// TIA Portal V15.1 export
// export: Created 2024-06-21T08:40:59.9132549Z, ExportSetting WithDefaults, DisplayName Totally Integrated Automation Portal, DisplayVersion V15.1 Update 5, DisplayName TIA Portal Openness, DisplayVersion V15.1 Update 5, DisplayName SINAMICS Startdrive Advanced, DisplayVersion V15.1, DisplayName G130, G150, S120, S150, SINAMICS MV, S210, DisplayVersion V15.1, DisplayName G110M, G120, G120C, G120D, G120P, DisplayVersion V15.1, DisplayName STEP 7 Professional, DisplayVersion V15.1 Update 5, DisplayName STEP 7 Safety, DisplayVersion V15.1, DisplayName WinCC Professional, DisplayVersion V15.1 Update 5, DisplayName SIMATIC Visualization Architect, DisplayVersion V15.1
FUNCTION_BLOCK "LPNIODiagHMIS7-1500"   // FB2214, FBD
TITLE = LPNIODiagHMIS7-1500
{ S7_Optimized_Access := 'FALSE' }
VERSION : 0.1
// stored: AutoNumber false, IsIECCheckEnabled false, SetENOAutomatically False, UDAEnableTagReadback false
   VAR_INPUT
      I_DeviceNumber { ExternalAccessible := 'False'; ExternalVisible := 'False'; ExternalWritable := 'False'} : Int;   // Device number in the hardware config
      I_Name { ExternalAccessible := 'False'; ExternalVisible := 'False'; ExternalWritable := 'False'} : String[25];   // Name device from list
      I_IPAddress { ExternalAccessible := 'False'; ExternalVisible := 'False'; ExternalWritable := 'False'} : String[15];   // IP address device from list
      I_MACAddress { ExternalAccessible := 'False'; ExternalVisible := 'False'; ExternalWritable := 'False'} : String[18];   // MAC address device from list
      I_AlarmClass { ExternalAccessible := 'False'; ExternalVisible := 'False'; ExternalWritable := 'False'} : Char;   // Alarm class -> A - B - C - D or E
      I_EnableAlarm { ExternalAccessible := 'False'; ExternalVisible := 'False'; ExternalWritable := 'False'} : Bool := TRUE;   // Enable alarm from upper level
      I_EnableButtons { ExternalAccessible := 'False'; ExternalVisible := 'False'; ExternalWritable := 'False'} : Bool;   // Enable to use the buttons in the pop-up -> "Activate" and "Deactivate"
   END_VAR
   VAR_OUTPUT
      O_Alarm { ExternalAccessible := 'False'; ExternalVisible := 'False'; ExternalWritable := 'False'} : Bool;   // Alarm A
      O_AC_Faulty { ExternalAccessible := 'False'; ExternalVisible := 'False'; ExternalWritable := 'False'} : Bool;   // Device is in faulty
      O_AD_Disabled { ExternalAccessible := 'False'; ExternalVisible := 'False'; ExternalWritable := 'False'} : Bool;   // Device is disabled
      O_AlarmABcondition { ExternalAccessible := 'False'; ExternalVisible := 'False'; ExternalWritable := 'False'} : Bool;   // Alarm AB condition
      H_IAnim { ExternalAccessible := 'False'; ExternalVisible := 'False'; ExternalWritable := 'False'} : Word;   // HMI Animation color of the icon
      H_IAnim2 { ExternalAccessible := 'False'; ExternalVisible := 'False'; ExternalWritable := 'False'} : Int;   // HMI Animation
   END_VAR
   VAR_IN_OUT
      IO_PNIODIAG_Global : "H_PNIODiagS7-1500";
   END_VAR
   VAR DB_SPECIFIC
      H_In : Struct   // HMI
         HMICmd : Word;   // Commands from HMI
         Mode : Int;   // Mode
      END_STRUCT;
      H_Out : Struct   // HMI
         Anim : Word;   // HMI Animation Word
         DeviceNumber : Int;   // HMI Device number (node)
         "Name" : String[25];   // HMI Profinet name
         IPAddress : String[15];   // HMI IP Address
         MACAddress : String[18];   // HMI MAC Address
         DBnr : Int;   // HMI Animation DB number
      END_STRUCT;
      HMICmdActivated { ExternalAccessible := 'False'; ExternalVisible := 'False'; ExternalWritable := 'False'} : Bool;   // HMI Cmd
      HMICmdDeactivated { ExternalAccessible := 'False'; ExternalVisible := 'False'; ExternalWritable := 'False'} : Bool;   // HMI Cmd
      Alarm { ExternalAccessible := 'False'; ExternalVisible := 'False'; ExternalWritable := 'False'} : Bool;   // Alarm
      AlarmClass_A { ExternalAccessible := 'False'; ExternalVisible := 'False'; ExternalWritable := 'False'} : Bool;   // The alarm is from alarm class A
      AlarmClass_B { ExternalAccessible := 'False'; ExternalVisible := 'False'; ExternalWritable := 'False'} : Bool;   // The alarm is from alarm class B
      AlarmClass_C { ExternalAccessible := 'False'; ExternalVisible := 'False'; ExternalWritable := 'False'} : Bool;   // The alarm is from alarm class C
      AlarmClass_D { ExternalAccessible := 'False'; ExternalVisible := 'False'; ExternalWritable := 'False'} : Bool;   // The alarm is from alarm class D
      AlarmClass_E { ExternalAccessible := 'False'; ExternalVisible := 'False'; ExternalWritable := 'False'} : Bool;   // The alarm is from alarm class E
      AlarmCond { ExternalAccessible := 'False'; ExternalVisible := 'False'; ExternalWritable := 'False'} : Bool;   // Alarm condition
      DBnr { ExternalAccessible := 'False'; ExternalVisible := 'False'; ExternalWritable := 'False'} : Int;   // HMI DB number
      DeviceExist { ExternalAccessible := 'False'; ExternalVisible := 'False'; ExternalWritable := 'False'} : Bool;   // Device exist
      DeviceDisabled { ExternalAccessible := 'False'; ExternalVisible := 'False'; ExternalWritable := 'False'} : Bool;   // Device is disabled
      DeviceFaulty { ExternalAccessible := 'False'; ExternalVisible := 'False'; ExternalWritable := 'False'} : Bool;   // Device is in faulty
      DeviceServiceReq { ExternalAccessible := 'False'; ExternalVisible := 'False'; ExternalWritable := 'False'} : Bool;   // Device has a service request
      EnableBtnActivate { ExternalAccessible := 'False'; ExternalVisible := 'False'; ExternalWritable := 'False'} : Bool;   // Enable button in pop-up
      EnableBtnDeactivate { ExternalAccessible := 'False'; ExternalVisible := 'False'; ExternalWritable := 'False'} : Bool;   // Enable button in pop-up
      TimerDeviceDisabled { ExternalAccessible := 'False'; ExternalVisible := 'False'; ExternalWritable := 'False'; S7_SetPoint := 'True'} : TOF_TIME;   // Timer
      TimerActivateDeactivateBusy { ExternalAccessible := 'False'; ExternalVisible := 'False'; ExternalWritable := 'False'; S7_SetPoint := 'True'} : TOF_TIME;   // Timer
      TimerHMICmdActivated { ExternalAccessible := 'False'; ExternalVisible := 'False'; ExternalWritable := 'False'; S7_SetPoint := 'True'} : TON_TIME;   // Timer
      TimerHMICmdDeactivated { ExternalAccessible := 'False'; ExternalVisible := 'False'; ExternalWritable := 'False'; S7_SetPoint := 'True'} : TON_TIME;   // Timer
   END_VAR
BEGIN

NETWORK
TITLE = **** 1 - Inputs **** DB number
// DB number
      L     DINO;
      T     #DBnr;

NETWORK
TITLE = **** 1 - Inputs **** Alarm class
// Alarm class
// Alarm class = E
      L     #I_AlarmClass;
      L     'E';
      ==I;
      =     #AlarmClass_E;

// Alarm class = D
      L     #I_AlarmClass;
      L     'D';
      ==I;
      =     #AlarmClass_D;

// Alarm class = C
      L     #I_AlarmClass;
      L     'C';
      ==I;
      =     #AlarmClass_C;

// Alarm class = B
      L     #I_AlarmClass;
      L     'B';
      ==I;
      =     #AlarmClass_B;

// Alarm class = A
      AN    #AlarmClass_B;
      AN    #AlarmClass_C;
      AN    #AlarmClass_D;
      AN    #AlarmClass_E;
      =     #AlarmClass_A;


REGION Network 3: **** 1 - Inputs **** HMI Cmd
   // Extract HMI Cmd
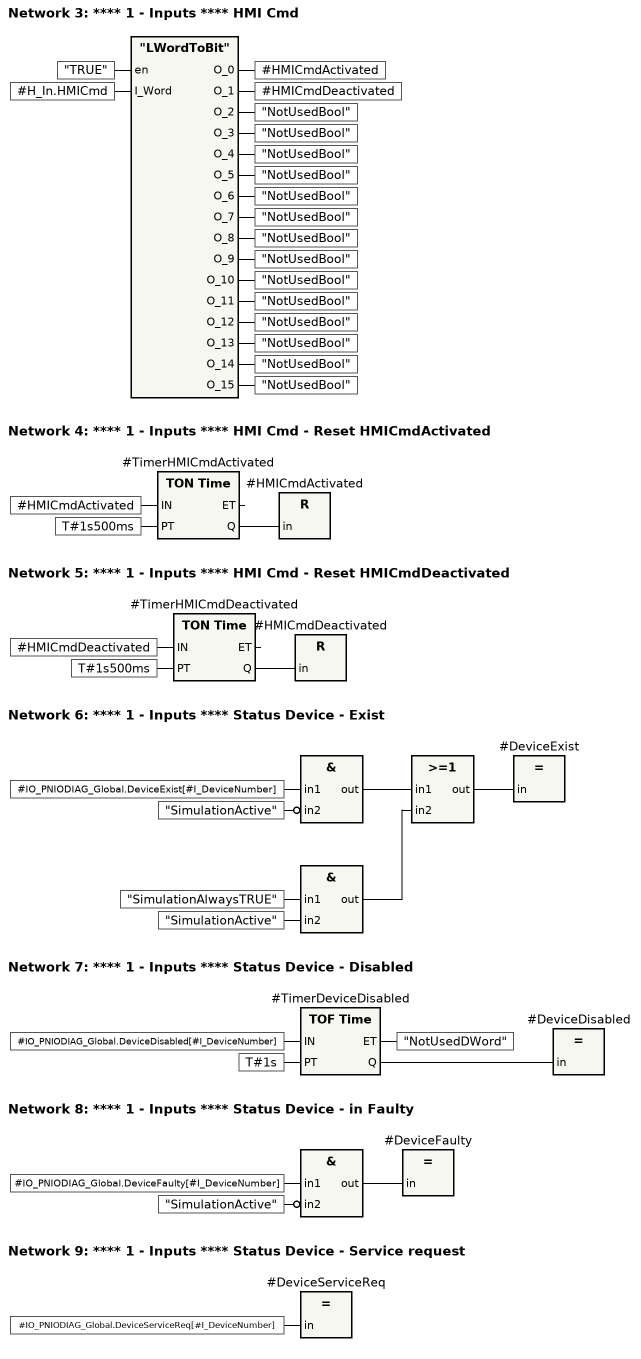
   IF "TRUE" THEN
       "LWordToBit"(I_Word := #H_In.HMICmd,
                    O_0 => #HMICmdActivated,
                    O_1 => #HMICmdDeactivated,
                    O_2 => "NotUsedBool",
                    O_3 => "NotUsedBool",
                    O_4 => "NotUsedBool",
                    O_5 => "NotUsedBool",
                    O_6 => "NotUsedBool",
                    O_7 => "NotUsedBool",
                    O_8 => "NotUsedBool",
                    O_9 => "NotUsedBool",
                    O_10 => "NotUsedBool",
                    O_11 => "NotUsedBool",
                    O_12 => "NotUsedBool",
                    O_13 => "NotUsedBool",
                    O_14 => "NotUsedBool",
                    O_15 => "NotUsedBool");
   END_IF;
END_REGION

REGION Network 4: **** 1 - Inputs **** HMI Cmd - Reset HMICmdActivated
   // HMI Cmd - Reset HMICmdActivated
   #TimerHMICmdActivated(IN := #HMICmdActivated, PT := T#1s500ms);   // TON
   IF #TimerHMICmdActivated.Q THEN #HMICmdActivated := FALSE; END_IF;
END_REGION

REGION Network 5: **** 1 - Inputs **** HMI Cmd - Reset HMICmdDeactivated
   // HMI Cmd - Reset HMICmdDeactivated
   #TimerHMICmdDeactivated(IN := #HMICmdDeactivated, PT := T#1s500ms);   // TON
   IF #TimerHMICmdDeactivated.Q THEN #HMICmdDeactivated := FALSE; END_IF;
END_REGION

REGION Network 6: **** 1 - Inputs **** Status Device - Exist
   // Status Device - Exist
   #DeviceExist := (#IO_PNIODIAG_Global.DeviceExist[#I_DeviceNumber] AND NOT "SimulationActive") OR ("SimulationAlwaysTRUE" AND "SimulationActive");
END_REGION

REGION Network 7: **** 1 - Inputs **** Status Device - Disabled
   // Status Device - Disabled
   #TimerDeviceDisabled(IN := #IO_PNIODIAG_Global.DeviceDisabled[#I_DeviceNumber],   // TOF
                        PT := T#1s,
                        ET => "NotUsedDWord");
   #DeviceDisabled := #TimerDeviceDisabled.Q;
END_REGION

REGION Network 8: **** 1 - Inputs **** Status Device - in Faulty
   // Status Device - in Faulty
   #DeviceFaulty := #IO_PNIODIAG_Global.DeviceFaulty[#I_DeviceNumber] AND NOT "SimulationActive";
END_REGION

REGION Network 9: **** 1 - Inputs **** Status Device - Service request
   // Status Device - Service request
   #DeviceServiceReq := #IO_PNIODIAG_Global.DeviceServiceReq[#I_DeviceNumber];
END_REGION

REGION Network 10: **** 1 - Inputs **** Timer Signal ActivateDeactivateBusy
   // Timer Signal ActivateDeactivateBusy
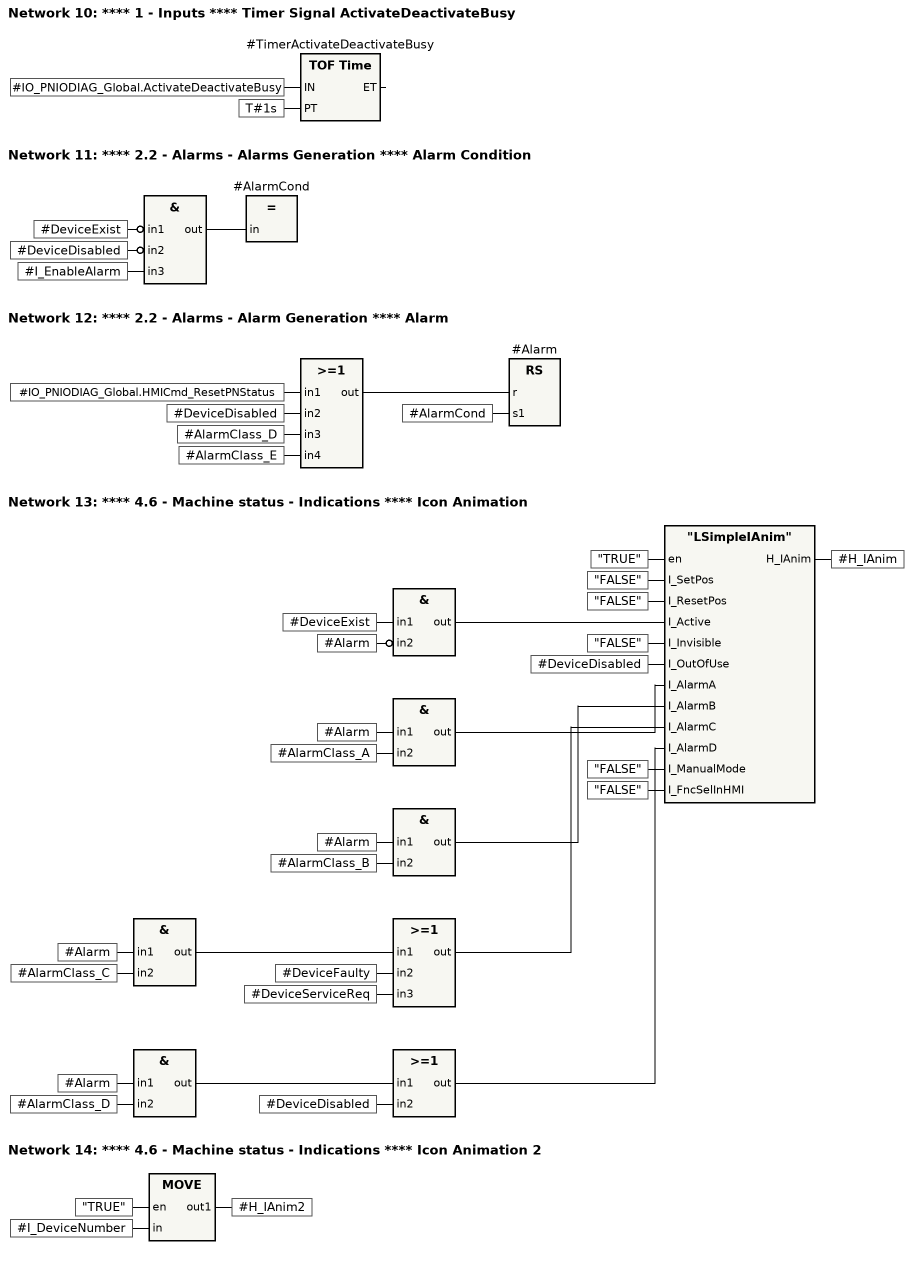
   #TimerActivateDeactivateBusy(IN := #IO_PNIODIAG_Global.ActivateDeactivateBusy, PT := T#1s);   // TOF
END_REGION

REGION Network 11: **** 2.2 - Alarms - Alarms Generation **** Alarm Condition
   // Condition for the Alarm
   #AlarmCond := NOT #DeviceExist AND NOT #DeviceDisabled AND #I_EnableAlarm;
END_REGION

REGION Network 12: **** 2.2 - Alarms - Alarm Generation **** Alarm
   // Alarm
   IF #IO_PNIODIAG_Global.HMICmd_ResetPNStatus OR #DeviceDisabled OR #AlarmClass_D OR #AlarmClass_E THEN
       #Alarm := FALSE;   // RS flip-flop
   END_IF;
   IF #AlarmCond THEN #Alarm := TRUE; END_IF;
END_REGION

REGION Network 13: **** 4.6 - Machine status - Indications **** Icon Animation
   // Icon Animation
   IF "TRUE" THEN
       "LSimpleIAnim"(I_SetPos := "FALSE",
                      I_ResetPos := "FALSE",
                      I_Active := #DeviceExist AND NOT #Alarm,
                      I_Invisible := "FALSE",
                      I_OutOfUse := #DeviceDisabled,
                      I_AlarmA := #Alarm AND #AlarmClass_A,
                      I_AlarmB := #Alarm AND #AlarmClass_B,
                      I_AlarmC := (#Alarm AND #AlarmClass_C) OR #DeviceFaulty OR #DeviceServiceReq,
                      I_AlarmD := (#Alarm AND #AlarmClass_D) OR #DeviceDisabled,
                      I_ManualMode := "FALSE",
                      I_FncSelInHMI := "FALSE",
                      H_IAnim => #H_IAnim);
   END_IF;
END_REGION

REGION Network 14: **** 4.6 - Machine status - Indications **** Icon Animation 2
   // Icon Animation Device number
   IF "TRUE" THEN #H_IAnim2 := #I_DeviceNumber; END_IF;
END_REGION

REGION Network 15: **** 4.6 - Machine status - Indications **** Animation
   // Animation for HMI
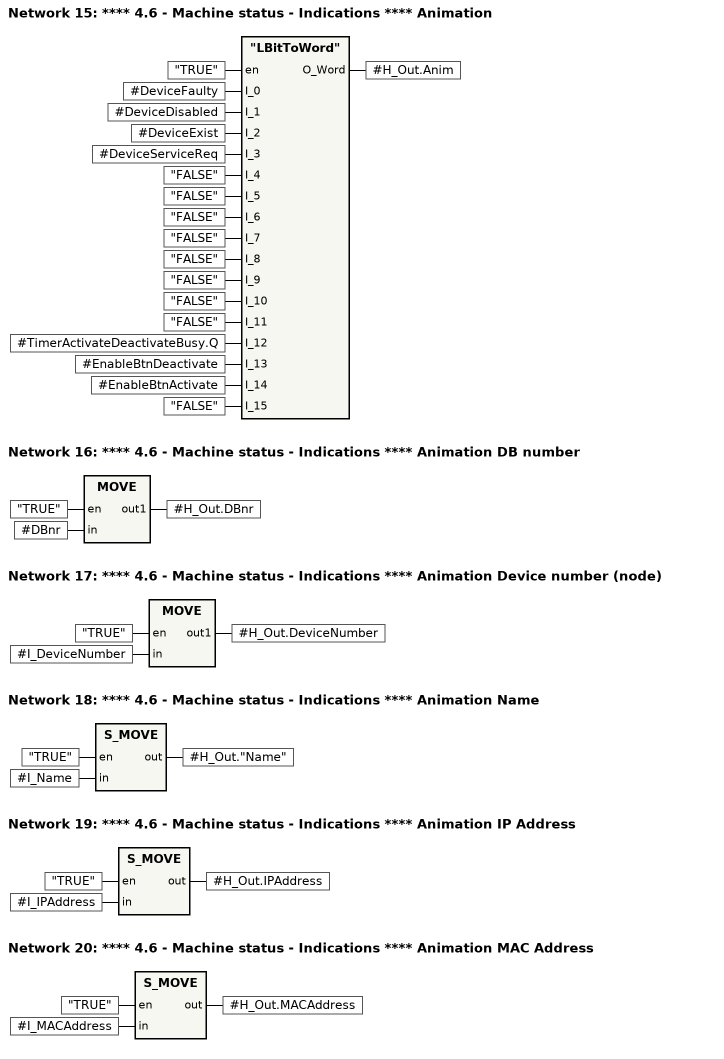
   IF "TRUE" THEN
       "LBitToWord"(I_0 := #DeviceFaulty,
                    I_1 := #DeviceDisabled,
                    I_2 := #DeviceExist,
                    I_3 := #DeviceServiceReq,
                    I_4 := "FALSE",
                    I_5 := "FALSE",
                    I_6 := "FALSE",
                    I_7 := "FALSE",
                    I_8 := "FALSE",
                    I_9 := "FALSE",
                    I_10 := "FALSE",
                    I_11 := "FALSE",
                    I_12 := #TimerActivateDeactivateBusy.Q,
                    I_13 := #EnableBtnDeactivate,
                    I_14 := #EnableBtnActivate,
                    I_15 := "FALSE",
                    O_Word => #H_Out.Anim);
   END_IF;
END_REGION

REGION Network 16: **** 4.6 - Machine status - Indications **** Animation DB number
   // DB number
   IF "TRUE" THEN #H_Out.DBnr := #DBnr; END_IF;
END_REGION

REGION Network 17: **** 4.6 - Machine status - Indications **** Animation Device number (node)
   // Device number (node)
   IF "TRUE" THEN #H_Out.DeviceNumber := #I_DeviceNumber; END_IF;
END_REGION

REGION Network 18: **** 4.6 - Machine status - Indications **** Animation Name
   // Name
   IF "TRUE" THEN #H_Out."Name" := #I_Name; END_IF;
END_REGION

REGION Network 19: **** 4.6 - Machine status - Indications **** Animation IP Address
   // IP Address
   IF "TRUE" THEN #H_Out.IPAddress := #I_IPAddress; END_IF;
END_REGION

REGION Network 20: **** 4.6 - Machine status - Indications **** Animation MAC Address
   // MAC Address
   IF "TRUE" THEN #H_Out.MACAddress := #I_MACAddress; END_IF;
END_REGION

REGION Network 21: **** 5.2 - Equations - Flow **** Activated or Deactived a device to the global FB
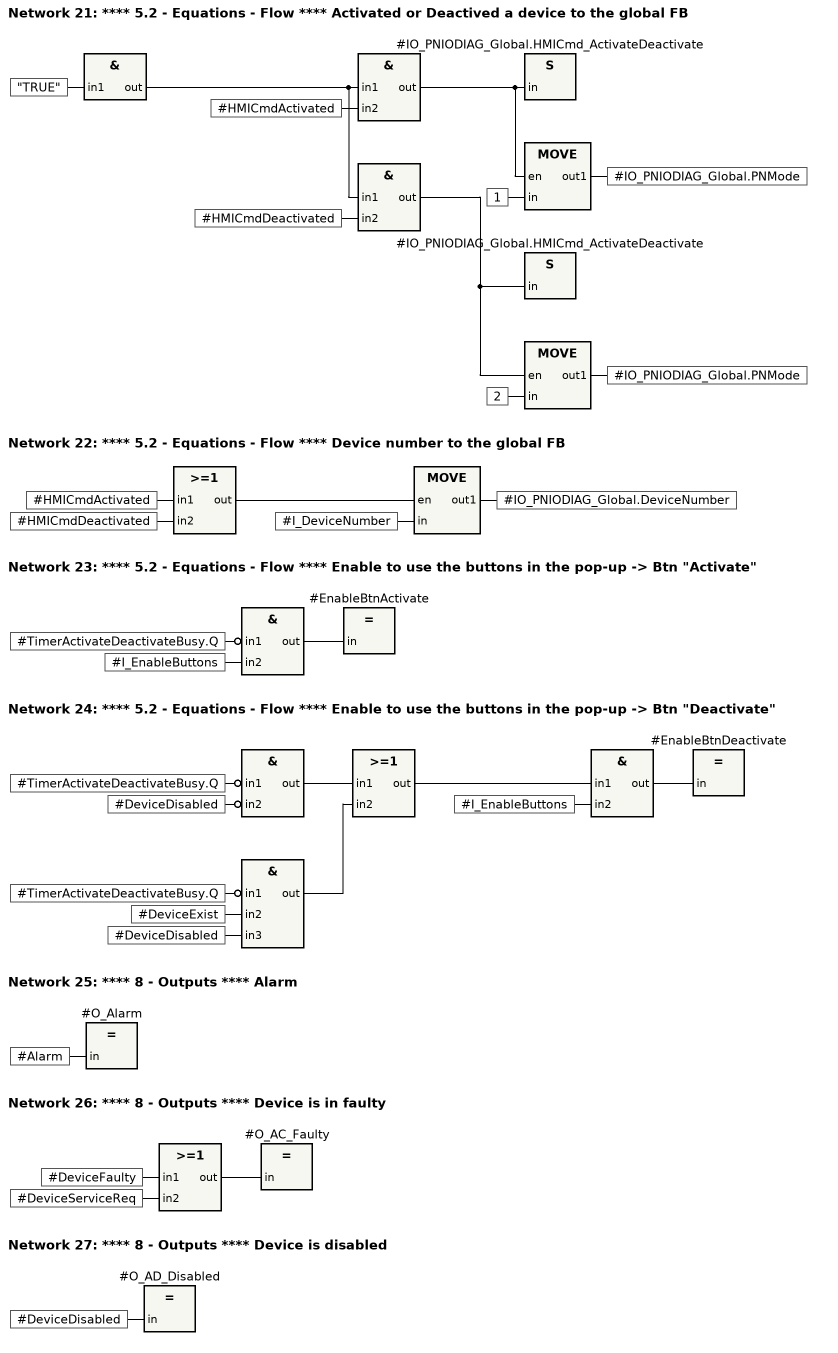
   IF "TRUE" AND #HMICmdActivated THEN
       #IO_PNIODIAG_Global.HMICmd_ActivateDeactivate := TRUE;
       #IO_PNIODIAG_Global.PNMode := 1;
   END_IF;
   IF "TRUE" AND #HMICmdDeactivated THEN
       #IO_PNIODIAG_Global.HMICmd_ActivateDeactivate := TRUE;
       #IO_PNIODIAG_Global.PNMode := 2;
   END_IF;
END_REGION

REGION Network 22: **** 5.2 - Equations - Flow **** Device number to the global FB
   IF #HMICmdActivated OR #HMICmdDeactivated THEN
       #IO_PNIODIAG_Global.DeviceNumber := #I_DeviceNumber;
   END_IF;
END_REGION

REGION Network 23: **** 5.2 - Equations - Flow **** Enable to use the buttons in the pop-up -> Btn "Activate"
   // Enable to use the buttons in the pop-up -> Btn "Activate"
   #EnableBtnActivate := NOT #TimerActivateDeactivateBusy.Q AND #I_EnableButtons;
END_REGION

REGION Network 24: **** 5.2 - Equations - Flow **** Enable to use the buttons in the pop-up -> Btn "Deactivate"
   // Enable to use the buttons in the pop-up -> Btn "Deactivate"
   #EnableBtnDeactivate := ((NOT #TimerActivateDeactivateBusy.Q AND NOT #DeviceDisabled) OR (NOT #TimerActivateDeactivateBusy.Q AND #DeviceExist AND #DeviceDisabled)) AND #I_EnableButtons;
END_REGION

REGION Network 25: **** 8 - Outputs **** Alarm
   // Alarm
   #O_Alarm := #Alarm;
END_REGION

REGION Network 26: **** 8 - Outputs **** Device is in faulty
   #O_AC_Faulty := #DeviceFaulty OR #DeviceServiceReq;
END_REGION

REGION Network 27: **** 8 - Outputs **** Device is disabled
   #O_AD_Disabled := #DeviceDisabled;
END_REGION

REGION Network 28: **** 8 - Outputs **** Alarm AB Condition
   // Alarm AB condition
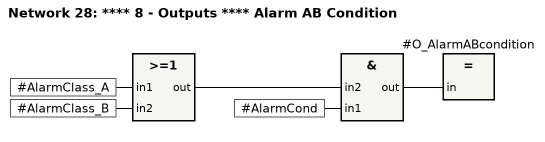
   #O_AlarmABcondition := (#AlarmClass_A OR #AlarmClass_B) AND #AlarmCond;
END_REGION
END_FUNCTION_BLOCK
